TYPE TcoDatamanUserData_v_5_x_x : STRUCT
    UserDataOption AT %Q* : UINT;
    UserDataLength AT %Q* : UINT;
    UserData AT %Q* : ARRAY[0..249] OF BYTE;
END_STRUCT
END_TYPE

(* stored: Version 1.1.0.1, ProductVersion 3.1.4024.11
   DUT TcoDatamanUserData_v_5_x_x: Id {402103af-ceb8-4f65-9e53-bac7c593eb57} *)
